SUBAPPLICATION Uebung_232_AX (* 2 ASRT-Quellen (Taster Last-Wins + echter Toggle-Taster) auf 1 ASRT-Latch via ASRT_MERGE_2, Ausgang Q1 *)
  (* Standard: 61499-2; Description: Copyright (c) 2026 Meisterschulen am Ostbahnhof This program and the accompanying materials are made available under the terms of the Eclipse Public License 2.0 which is available at https://www.eclipse.org/legal/epl-2.0/ SPDX-License-Identifier: EPL-2.0 *)
  (* Version 1.0, 2026-09-06, Franz Höpfinger, Meisterschulen am Ostbahnhof, initial API and implementation and/or initial documentation *)
  PACKAGE Uebungen;
  IMPORT logiBUS::io::DI::logiBUS_DI::Input_I1;
  IMPORT logiBUS::io::DI::logiBUS_DI::Input_I2;
  IMPORT logiBUS::io::DI::logiBUS_DI_Events::BUTTON_SINGLE_CLICK;
  IMPORT logiBUS::io::DQ::logiBUS_DO::Output_Q1;
  (* Documentation:
  2 ASRT-Quellen ODER-verknüpft auf 1 ASRT-Latch
   Direktes Geschwister zu Uebung_229_AX/Uebung_230_AX, aber mit ASRT (Set/Reset/Toggle) statt ASR (nur Set/Reset) durchgängig: zwei unabhängige Quellen liefern je einen Teil der SET/RESET/TOGGLE-Semantik, ASRT_MERGE_2 führt beide zu einem gemeinsamen ASRT_AX_T_FF_SR-Latch zusammen.
   Funktionsbeschreibung
    - Quelle 1 (AX_ASRT_RF_TRIG): klassischer Taster an Input_I1. Drücken (steigende Flanke) → SET, Loslassen (fallende Flanke) → RESET. TOGGLE feuert hier nie - aus einem reinen Flankensignal lässt sich kein drittes, unabhängiges Ereignis ableiten.
   - Quelle 2 (ASRT_3EVENTS_TO_SRT): ein waschechter Toggle-Taster an Input_I2 (BUTTON_SINGLE_CLICK) - hier ist nur TOGGLE verdrahtet, SET/RESET bleiben unbenutzt.
   - ASRT_MERGE_2 vereinigt beide Streams zu einem gemeinsamen ASRT-Signal, bevor es auf ASRT_AX_T_FF_SR.S_R_T trifft - dieselbe ODER-Zusammenführung wie bei ASR_MERGE_2 in Uebung_230_AX, jetzt eben inklusive der dritten (Toggle-)Schiene.
    Arbeitsauftrag
   Testen Sie: Taster I1 drücken und halten → Q1 EIN, solange gedrückt (Last-Wins wie in 229/230). Taster I1 loslassen → Q1 AUS. Unabhängig davon jederzeit den Toggle-Taster I2 klicken → Q1 wechselt seinen aktuellen Zustand, egal was I1 gerade macht.
   Referenzlösung
   Uebung_232_AX.SUB. Der neue Baustein AX_ASRT_RF_TRIG liegt als Composite-SubApp in MyLib_AX-1.0.0/typelib/sys/AX_ASRT_RF_TRIG.SUB - aus dem bestehenden AX_ASR_RF_TRIG plus ASRT_SR_AE_TO_SRT (SR_IN direkt aus dem ASR, TOGGLE_IN unverdrahtet), statt eines neuen Low-Level-FBTypes.
  *)
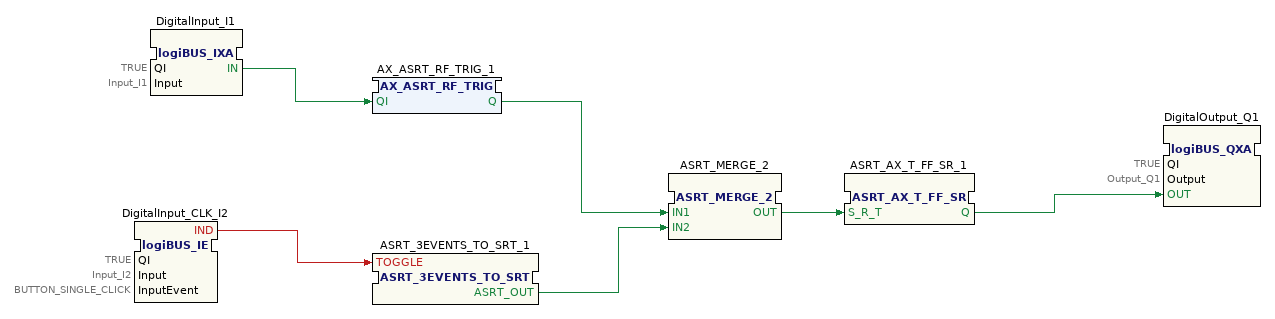
  (* Quelle 1 (AX_ASRT_RF_TRIG): Taster gedrueckt=SET, losgelassen=RESET - TOGGLE bleibt ungenutzt. Quelle 2 (ASRT_3EVENTS_TO_SRT): nur TOGGLE verdrahtet, SET/RESET bleiben offen - ein echter Taster mit Klick-Umschaltung. ASRT_MERGE_2 fuehrt beide ASRT-Streams zusammen, bevor sie auf denselben ASRT_AX_T_FF_SR treffen. *)
  FBS
    DigitalInput_I1 : logiBUS::io::DI::logiBUS_IXA(QI := TRUE, Input := Input_I1);
    DigitalInput_CLK_I2 : logiBUS::io::DI::logiBUS_IE(QI := TRUE, Input := Input_I2, InputEvent := BUTTON_SINGLE_CLICK);
    ASRT_3EVENTS_TO_SRT_1 : adapter::conversion::unidirectional::ASRT_3EVENTS_TO_SRT;
    ASRT_MERGE_2 : adapter::events::unidirectional::ASRT_MERGE_2;
    ASRT_AX_T_FF_SR_1 : adapter::events::unidirectional::ASRT_AX_T_FF_SR;
    DigitalOutput_Q1 : logiBUS::io::DQ::logiBUS_QXA(QI := TRUE, Output := Output_Q1);
  END_FBS
  SUBAPPS
    AX_ASRT_RF_TRIG_1 : MyLib::sys::AX_ASRT_RF_TRIG;
  END_SUBAPPS
  EVENT_CONNECTIONS
    DigitalInput_CLK_I2.IND TO ASRT_3EVENTS_TO_SRT_1.TOGGLE;
  END_CONNECTIONS
  ADAPTER_CONNECTIONS
    DigitalInput_I1.IN TO AX_ASRT_RF_TRIG_1.QI;
    AX_ASRT_RF_TRIG_1.Q TO ASRT_MERGE_2.IN1;
    ASRT_3EVENTS_TO_SRT_1.ASRT_OUT TO ASRT_MERGE_2.IN2;
    ASRT_MERGE_2.OUT TO ASRT_AX_T_FF_SR_1.S_R_T;
    ASRT_AX_T_FF_SR_1.Q TO DigitalOutput_Q1.OUT;
  END_CONNECTIONS
END_SUBAPPLICATION
